FUNCTION_BLOCK InputDecompressor (* Basic Function Block Type *)
  (* Standard: 61499-2 *)
  (* Version 0.0, 6/21/2018, Rediska, nxtControl GmbH, Template *)
  PACKAGE Main;
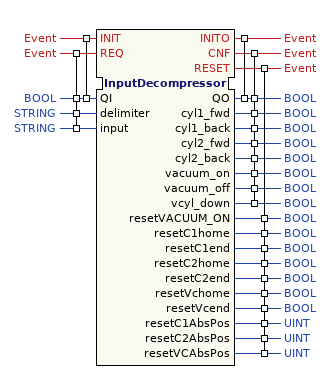
  EVENT_INPUT
    INIT WITH QI; (* Initialization Request *)
    REQ WITH QI, delimiter, input; (* Normal Execution Request *)
  END_EVENT
  EVENT_OUTPUT
    INITO WITH QO; (* Initialization Confirm *)
    CNF WITH QO, cyl1_fwd, cyl1_back, cyl2_fwd, cyl2_back, vacuum_on, vacuum_off, vcyl_down; (* Execution Confirmation *)
    RESET WITH resetVACUUM_ON, resetC1home, resetC1end, resetC2home, resetC2end, resetVchome, resetVcend, resetC1AbsPos, resetC2AbsPos, resetVCAbsPos;
  END_EVENT
  VAR_INPUT
    QI : BOOL; (* Input event qualifier *)
    delimiter : STRING;
    input : STRING;
  END_VAR
  VAR_OUTPUT
    QO : BOOL; (* Output event qualifier *)
    cyl1_fwd : BOOL;
    cyl1_back : BOOL;
    cyl2_fwd : BOOL;
    cyl2_back : BOOL;
    vacuum_on : BOOL;
    vacuum_off : BOOL;
    vcyl_down : BOOL;
    resetVACUUM_ON : BOOL;
    resetC1home : BOOL;
    resetC1end : BOOL;
    resetC2home : BOOL;
    resetC2end : BOOL;
    resetVchome : BOOL;
    resetVcend : BOOL;
    resetC1AbsPos : UINT;
    resetC2AbsPos : UINT;
    resetVCAbsPos : UINT;
  END_VAR
  VAR
    reset : BOOL;
    subs : ARRAY [0..22] OF STRING;
  END_VAR
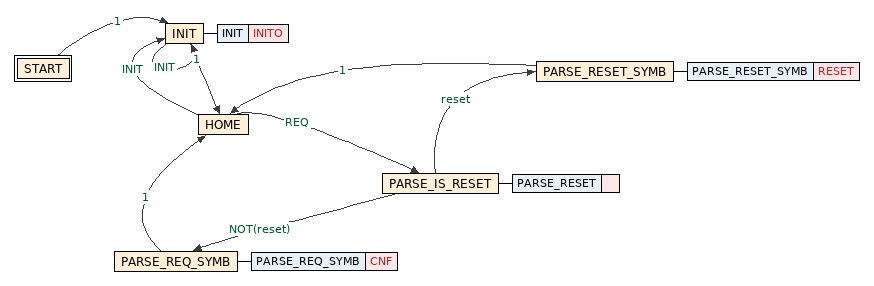
  EC_STATES
    START; (* Initial State *)
    INIT : INIT -> INITO; (* Initialization *)
    PARSE_IS_RESET : PARSE_RESET;
    PARSE_RESET_SYMB : PARSE_RESET_SYMB -> RESET;
    PARSE_REQ_SYMB : PARSE_REQ_SYMB -> CNF;
    HOME;
  END_STATES
  EC_TRANSITIONS
    START TO INIT := 1;
    HOME TO PARSE_IS_RESET := REQ;
    PARSE_IS_RESET TO PARSE_REQ_SYMB := NOT(reset);
    PARSE_REQ_SYMB TO HOME := 1;
    PARSE_RESET_SYMB TO HOME := 1;
    PARSE_IS_RESET TO PARSE_RESET_SYMB := reset;
    INIT TO INIT := INIT;
    INIT TO HOME := 1;
    HOME TO INIT := INIT;
  END_TRANSITIONS
  ALGORITHM INIT IN ST: (* Initialization algorithm *)
QO := TRUE;
INIT:=FALSE;
  END_ALGORITHM
  ALGORITHM REQ IN ST: (* Normally executed algorithm *)
;
  END_ALGORITHM
  ALGORITHM PARSE_RESET_SYMB IN ST:
VAR
	length: INT;
	i : INT;
	prev: INT;
	substr : ARRAY[1..11] OF STRING;
	num : INT;
	cur: INT;
END_VAR;
length := DINT_TO_INT(LEN(input));
prev := 1;
cur := 1;
FOR i := 1 TO length DO
	IF (MID(input,1,i) = delimiter) THEN

		substr[cur] := MID(input, i - prev, prev);//input.DATA[prev, i-1];
		cur := cur + 1;
		prev := i + 1;
	END_IF;
END_FOR;
resetVACUUM_ON := STRING_TO_BOOL(substr[2]);
resetC1home := STRING_TO_BOOL(substr[3]);
resetC1end := STRING_TO_BOOL(substr[4]);

resetC2home := STRING_TO_BOOL(substr[5]);
resetC2end := STRING_TO_BOOL(substr[6]);
resetVchome := STRING_TO_BOOL(substr[7]);
resetVcend := STRING_TO_BOOL(substr[8]);

resetC1AbsPos := STRING_TO_UINT(substr[9]);
resetC2AbsPos := STRING_TO_UINT(substr[10]);
resetVCAbsPos := STRING_TO_UINT(substr[11]);
  END_ALGORITHM
  ALGORITHM PARSE_REQ_SYMB IN ST:
VAR
	length: INT;
	i : INT;
	prev: INT;
	substr : ARRAY[1..8] OF STRING;
	num : INT;
	cur: INT;
END_VAR;
length := DINT_TO_INT(LEN(input));
prev := 1;
cur := 1;
FOR i := 1 TO length DO
	IF (MID(input,1,i) = delimiter) THEN
		substr[cur] := MID(input, i - prev, prev);//input.DATA[prev, i-1];
		cur := cur + 1;
		prev := i + 1;
	END_IF;
END_FOR;
cyl1_fwd := STRING_TO_BOOL(substr[2]);
cyl1_back := STRING_TO_BOOL(substr[3]);
cyl2_fwd := STRING_TO_BOOL(substr[4]);
cyl2_back := STRING_TO_BOOL(substr[5]);
vacuum_on := STRING_TO_BOOL(substr[6]);
vacuum_off := STRING_TO_BOOL(substr[7]);
vcyl_down := STRING_TO_BOOL(substr[8]);
  END_ALGORITHM
  ALGORITHM PARSE_RESET IN ST:
VAR
	i: INT;
END_VAR;
i := 1;
(*WHILE MID(input, 1, i) <> delimiter DO
	i := i + 1;
END_WHILE;*)
INIT:=FALSE;
reset := STRING_TO_BOOL(MID(input, i, 1));
  END_ALGORITHM
END_FUNCTION_BLOCK
